PROGRAM pouMachineSettings
VAR
	btnOSRRead:R_TRIG;
	btnOSRWrite:R_TRIG;
	
	
    fbFileOpen           : FB_FileOpen;
    fbFileClose          : FB_FileClose;
    fbFileRead           : FB_FileRead;
    fbFileWrite          : FB_FileWrite;
    hFile             : UINT := 0;(* File handle of the source file *)
 	strFilePath:STRING := 'C:\PLC\testfile.txt';
	
	strSampleString:STRING :='This is my sample string, and this is some more text';
	
	
	

END_VAR


//capture OSR for buttons
btnOSRRead	(	CLK := MachineSettings.btnRead);
btnOSRWrite	(	CLK := MachineSettings.btnWrite);


actWriteFile();

ACTION actWriteFile:

//create handle
fbFileOpen(sNetId :=,
			sPathName :=strFilePath,
			nMode :=FOPEN_MODEWRITE,
			ePath	:=PATH_GENERIC,
			bExecute :=btnOSRWrite.Q,
			tTimeout :=,
			);
	
			hFile := fbFileOpen.hFile;
		

//close handle			
IF hFile > 1 THEN
		
	//do somthing
	fbFileWrite(	sNetId:=,
					hFile := hFile,
					pWriteBuff:=ADR(strSampleString),
					cbWriteLen:=SIZEOF(strSampleString),
					bExecute:=TRUE,
					tTimeout:=,
					);
					
END_IF
				
	fbFileWrite( bExecute := FALSE);
			




//close handle			
IF hFile > 1 THEN
	
fbFileClose(sNetId:=,
			hFile:=hFile,
			bExecute:=TRUE,
			tTimeout:=,
			);
			


END_IF


//reset handle
hFile := 0;


//close request to close handle
fbFileClose(bExecute:=FALSE);
END_ACTION

END_PROGRAM

(* stored: Version 1.1.0.1, ProductVersion 3.1.4024.11
   POU pouMachineSettings: Id {2c1d7b51-dab5-0b83-12e9-3cad039059fd}, SpecialFunc None
   Action actWriteFile: Id {599b32ba-5778-0bec-3bb7-ae7367022332} *)
